FUNCTION_BLOCK WARPPOLAR (* openCV warp polar *)
  (* Version 1.0, AN, SWDC RTSoft *)
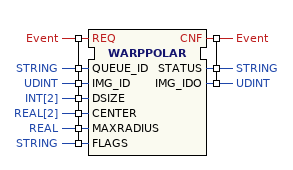
  EVENT_INPUT
    REQ WITH QUEUE_ID, IMG_ID, DSIZE, CENTER, MAXRADIUS, FLAGS;
  END_EVENT
  EVENT_OUTPUT
    CNF WITH STATUS, IMG_IDO;
  END_EVENT
  VAR_INPUT
    QUEUE_ID : STRING;
    IMG_ID : UDINT;
    DSIZE : ARRAY [0..1] OF INT; (* Size of the output image (width, height) *)
    CENTER : ARRAY [0..1] OF REAL; (* Center of the polar transformation (x, y) *)
    MAXRADIUS : REAL; (* Maximum radius of the polar transformation *)
    FLAGS : STRING;
  END_VAR
  VAR_OUTPUT
    STATUS : STRING;
    IMG_IDO : UDINT;
  END_VAR
  ALGORITHM REQ IN ST:

  END_ALGORITHM
END_FUNCTION_BLOCK
